KUKA KRL program: move_to_maintenance_pos.src, move_to_maintenance_pos.dat

--- move_to_maintenance_pos.src ---
&ACCESS RVO1
&REL 19
&PARAM EDITMASK = *
&PARAM TEMPLATE = C:\KRC\Roboter\Template\vorgabe
DEF move_to_maintenance_pos( )
   ;FOLD INI;%{PE}
      ;FOLD BASISTECH INI
         GLOBAL INTERRUPT DECL 3 WHEN $STOPMESS==TRUE DO IR_STOPM ( )
         INTERRUPT ON 3
         BAS (#INITMOV,0 )
      ;ENDFOLD (BASISTECH INI)
      ;FOLD USER INI
         ;Make your modifications here

      ;ENDFOLD (USER INI)
   ;ENDFOLD (INI)

   IF NOT $IN_HOME3 THEN
      move_to_perch_pos()
   ENDIF

;FOLD PTP home3 Vel=15 % PDAT2;%{PE}%R 8.3.38,%MKUKATPBASIS,%CMOVE,%VPTP,%P 1:PTP, 2:home3, 3:, 5:15, 7:PDAT2
$BWDSTART=FALSE
PDAT_ACT=PPDAT2
FDAT_ACT=Fhome3
BAS(#PTP_PARAMS,15)
PTP Xhome3
;ENDFOLD

   ;FOLD HandShake[5 : At Maintenance Position], WAIT on Response
;FOLD ;%{h}
;Params IlfProvider=model3_handshakectrl; Core_CmdTechHandShake=HandShake; Core_CmdHandShake=5; Core_Wait=True
;ENDFOLD
HandShake_Set (5,false)
HandShake_Check (5,false)
;ENDFOLD

   move_to_perch_pos()

END

--- move_to_maintenance_pos.dat ---
&ACCESS RVO1
&REL 19
&PARAM EDITMASK = *
&PARAM TEMPLATE = C:\KRC\Roboter\Template\vorgabe
DEFDAT  move_to_maintenance_pos
;FOLD EXTERNAL DECLARATIONS;%{PE}%MKUKATPBASIS,%CEXT,%VCOMMON,%P
;FOLD BASISTECH EXT;%{PE}%MKUKATPBASIS,%CEXT,%VEXT,%P
EXT  BAS (BAS_COMMAND  :IN,REAL  :IN )
DECL INT SUCCESS
;ENDFOLD (BASISTECH EXT)
;FOLD USER EXT;%{E}%MKUKATPUSER,%CEXT,%VEXT,%P
;Make your modifications here

;ENDFOLD (USER EXT)
;ENDFOLD (EXTERNAL DECLARATIONS)
DECL E6POS Xweld_pos={X -85.9545,Y -1068.13318,Z 1203.34253,A 9.17978477,B 0.595385969,C 45.0561867,S 6,T 18,E1 0.0,E2 0.0,E3 0.0,E4 0.0,E5 0.0,E6 0.0}
DECL FDAT Fweld_pos={TOOL_NO 1,BASE_NO 0,IPO_FRAME #BASE,POINT2[] " "}
DECL MODULEPARAM_T LAST_TP_PARAMS={PARAMS[] "Kuka.VelocityFieldEnabled=True; Kuka.ColDetectFieldEnabled=True; Kuka.MovementParameterFieldEnabled=True; Kuka.IsAngleEnabled=False; Kuka.PointName=weld_pos; Kuka.FrameData.base_no=0; Kuka.FrameData.tool_no=1; Kuka.FrameData.ipo_frame=#BASE; Kuka.FrameData.point2=; Kuka.isglobalpoint=False; Kuka.VelocityPtp=5; Kuka.BlendingEnabled=False; Kuka.CurrentCDSetIndex=0   "}
DECL FDAT FHOME2={TOOL_NO 1,BASE_NO 0,IPO_FRAME #BASE,POINT2[] " "}
DECL BASIS_SUGG_T LAST_BASIS={POINT1[] "home3                   ",POINT2[] "home3                   ",CP_PARAMS[] "CPDAT0                  ",PTP_PARAMS[] "PDAT2                   ",CONT[] "                        ",CP_VEL[] "2.0                     ",PTP_VEL[] "5                       ",SYNC_PARAMS[] "SYNCDAT                 ",SPL_NAME[] "S0                      ",A_PARAMS[] "ADAT0                   "}
DECL FDAT Fhome4={TOOL_NO 1,BASE_NO 0,IPO_FRAME #BASE,POINT2[] " ",TQ_STATE FALSE}
DECL PDAT PPDAT1={VEL 100.000,ACC 5.00000,APO_DIST 100.000,APO_MODE #CDIS,GEAR_JERK 50.0000,EXAX_IGN 0}
DECL FDAT Fhome3={TOOL_NO 1,BASE_NO 0,IPO_FRAME #BASE,POINT2[] " ",TQ_STATE FALSE}
DECL PDAT PPDAT2={VEL 100.000,ACC 5.00000,APO_DIST 100.000,APO_MODE #CDIS,GEAR_JERK 50.0000,EXAX_IGN 0}
ENDDAT
